IF (Uds_s.status = 1) THEN
	IF (Uds_s.status = 1 AND Uds_s.UdsTx.dataSize > 0) THEN
		IF (Uds_s.UdsTx.dataSize = Uds_s.UdsTx.data[1]) THEN (*send sf or ff*)
			IF (Uds_s.UdsTx.dataSize <= 7) THEN (*sf*)
				FOR y := 1 TO 8 DO
					tempCanSendBuff[y] := Uds_s.UdsTx.data[y];
				END_FOR
				IF (Uds_s.UdsTx.data[2] = 16#30) THEN
				can_sendDatabox(0, 42, Uds_s.UdsTx.dataSize, ADR(tempCanSendBuff) + 1);
				ELSE
				can_sendDatabox(0, 42, Uds_s.UdsTx.dataSize + 1, ADR(tempCanSendBuff));
				END_IF
				Uds_s.UdsTx.dataSize := 0;
				Uds_s.UdsTx.data[1] := 0;
			ELSE (*ff*)
				bytesTxFf[1] := 16#10;
				bytesTxFf[2] := Uds_s.UdsTx.data[1];
				FOR y := 3 TO 8 DO
					bytesTxFf[y] := Uds_s.UdsTx.data[y - 1];
				END_FOR
				Uds_s.UdsTx.data[1] := Uds_s.UdsTx.data[1] - 6;
				can_sendDatabox(0, 42, 8, ADR(bytesTxFf));
			END_IF
			Uds_s.status := 0;
		ELSIF (Uds_s.UdsTx.dataSize > Uds_s.UdsTx.data[1]) THEN (*cf*)
			startIndex := Uds_s.UdsTx.dataSize - Uds_s.UdsTx.data[1];
			bytesTxCf[1] := 16#20 + ((startIndex + 1) / 7) MOD 10;
			FOR txCfIdx := 2 TO 8 DO
				bytesTxCf[txCfIdx] := Uds_s.UdsTx.data[startIndex + txCfIdx];
				Uds_s.UdsTx.data[1] := Uds_s.UdsTx.data[1] - 1;
				IF (Uds_s.UdsTx.data[1] = 0) THEN
					EXIT;
				END_IF
			END_FOR
			IF (txCfIdx > 8) THEN
				txCfIdx := 8;
			END_IF
			can_sendDatabox(0, 42, txCfIdx, ADR(bytesTxCf));
			IF (Uds_s.UdsTx.data[1] = 0) THEN
				Uds_s.status := 0;
				Uds_s.UdsTx.dataSize := 0;
				Uds_s.UdsTx.data[1] := 0;
			END_IF
		END_IF
		Uds_s.tester := 0;
	END_IF
END_IF

IF (Uds_s.status = 0 AND Uds_s.UdsRx.data[1] = Uds_s.UdsRx.dataSize AND Uds_s.UdsRx.dataSize > 0) THEN
	Uds();
	Uds_s.UdsRx.dataSize := 0;
	Uds_s.UdsRx.data[1] := 0;
	Uds_s.status := 1;
END_IF
END_PROGRAM

(* POU Uds/Uds, ST *)
PROGRAM Uds
VAR
END_VAR
CASE Uds_s.UdsRx.data[2] OF
	16#10: UdsSrvDsc();
(*
	16#11: UdsSrvRst();*)
	16#14: UdsSrvClrDiagcInfo();

	16#19: UdsSrvReadDtcInfo();

	16#22: UdsSrvReadDataById();
(*
	16#23: UdsSrvReadMemByAddr();
	16#27: UdsSrvSecuAcs();*)
	16#2E: UdsSrvWriteDataById();
	(*16#31: UdsSrvRoutineCtrl();
	16#3D: UdsSrvWrMemByAddr();*)
	16#3E: UdsSrvTesterPresent();

ELSE
	UdsSrvNotSupported();
END_CASE;
END_PROGRAM

(* POU Uds/UdsSrvDsc, ST *)
PROGRAM UdsSrvDsc
VAR
END_VAR
IF (Uds_s.UdsRx.dataSize = 2 AND (Uds_s.UdsRx.data[3] = 16#01 OR Uds_s.UdsRx.data[3] = 16#03)) THEN
	Uds_s.sessionType := Uds_s.UdsRx.data[3];
	Uds_s.activeAccessLevel_u8 := LID_DevelopmentSession_DU8;(*LID_DefaultSession_DU8;*)
	Uds_s.UdsTx.dataSize := 6;
	Uds_s.UdsTx.data[1] := Uds_s.UdsTx.dataSize;
	Uds_s.UdsTx.data[2] := 16#50;
	Uds_s.UdsTx.data[3] := Uds_s.sessionType;
	Uds_s.UdsTx.data[4] := 16#00;
	Uds_s.UdsTx.data[5] := 16#96;
	Uds_s.UdsTx.data[6] := 16#01;
	Uds_s.UdsTx.data[7] := 16#F4;
ELSE
	UdsSrvNotSupported(); (*Temp solution, throw 7F error*)
END_IF
END_PROGRAM

(* POU Uds/UdsSrvNotSupported, ST *)
PROGRAM UdsSrvNotSupported
VAR
END_VAR
Uds_s.UdsTx.dataSize := 3;
Uds_s.UdsTx.data[1] := Uds_s.UdsTx.dataSize;
Uds_s.UdsTx.data[2] := 16#7F;
Uds_s.UdsTx.data[3] := Uds_s.UdsRx.data[3];
Uds_s.UdsTx.data[4] := 16#11;
END_PROGRAM

(* POU Uds/UdsSrvClrDiagcInfo, ST *)
PROGRAM UdsSrvClrDiagcInfo
VAR
	groupOfDtc : UDINT;
END_VAR
IF (Uds_s.UdsRx.dataSize = 4) THEN
	groupOfDtc := SHL(USINT_TO_UDINT(Uds_s.UdsRx.data[3]), 16);
	groupOfDtc := groupOfDtc + SHL(USINT_TO_UDINT(Uds_s.UdsRx.data[4]), 8);
	groupOfDtc := groupOfDtc + Uds_s.UdsRx.data[5];
	IF (groupOfDtc = 16#FFFFFF) THEN
		sys_enterCriticalSection();
		sys_delActiveErrors();
		sys_delSavedErrors();
		sys_leaveCriticalSection();
	END_IF
END_IF
END_PROGRAM

(* POU Uds/UdsSrvReadDtcInfo, ST *)
PROGRAM UdsSrvReadDtcInfo
VAR
	numSavedErr_u16        : UINT;
	numActvErr_u16         : UINT;
	numActvAndSavedErr_u16 : UINT;
	numErr_u16             : UINT;
	errData_s              : ErrorData_ts;
	idx_u16                : UINT;
	cntDtc_u16             : UINT;

	dtc_u32                : UDINT;
	dtcHB_u8               : USINT;
	dtcMB_u8               : USINT;
	dtcLB_u8               : USINT;

	buf_au8                : ARRAY[1..250] OF USINT; (*data without SID*)
	bufLength_u8           : USINT; (*actual data size*)
	i                      : USINT;
	idxErr_u8				  : USINT;
END_VAR
Uds_s.UdsTx.data[1] := 0;
IF (Uds_s.UdsRx.dataSize = 3) THEN
   IF (Uds_s.UdsRx.data[3] = 1) THEN
      sys_enterCriticalSection();
      IF (Uds_s.UdsRx.data[4] = 1) THEN
         numActvErr_u16 := sys_getNumActiveErrors();
      ELSIF (Uds_s.UdsRx.data[4] = 8) THEN
         numSavedErr_u16 := sys_getNumSavedErrors();
      END_IF
			IF (Uds_s.UdsRx.data[5] = 9) THEN
				WHILE(TRUE) DO
					numErr_u16 := sys_getSavedErrors( ADR(errData_s), idx_u16, 1);
				   IF numErr_u16 <> 1 THEN
					   EXIT;
				   END_IF

				   IF sys_testError(errData_s.Code_u16, errData_s.Param_u8) <> 0 THEN
					   numActvAndSavedErr_u16 := numActvAndSavedErr_u16 + 1;
				   END_IF
				   idx_u16 := idx_u16 + 1;
			   END_WHILE
			END_IF
		sys_leaveCriticalSection();
		IF ((numSavedErr_u16 + numActvErr_u16) >= numActvAndSavedErr_u16) THEN
			cntDtc_u16 := numSavedErr_u16 + numActvErr_u16 - numActvAndSavedErr_u16;
		ELSE
		   cntDtc_u16 := numSavedErr_u16 + numActvErr_u16;
	   END_IF

		Uds_s.UdsTx.data[1] := Uds_s.UdsTx.data[1] + 1;
		Uds_s.UdsTx.data[Uds_s.UdsTx.data[1] + 1 ] := Uds_s.UdsRx.data[2] + 16#40;
		Uds_s.UdsTx.data[1] := Uds_s.UdsTx.data[1] + 1;
		Uds_s.UdsTx.data[Uds_s.UdsTx.data[1] + 1 ] := Uds_s.UdsRx.data[3];
		Uds_s.UdsTx.data[1] := Uds_s.UdsTx.data[1] + 1;
		Uds_s.UdsTx.data[Uds_s.UdsTx.data[1] + 1 ] := Uds_s.UdsRx.data[4];
		Uds_s.UdsTx.data[1] := Uds_s.UdsTx.data[1] + 1;
		Uds_s.UdsTx.data[Uds_s.UdsTx.data[1] + 1 ] := Uds_s.UdsRx.data[5];
		Uds_s.UdsTx.data[1] := Uds_s.UdsTx.data[1] + 1;
		Uds_s.UdsTx.data[Uds_s.UdsTx.data[1] + 1 ] := UINT_TO_USINT(SHR(cntDtc_u16, 8));
		Uds_s.UdsTx.data[1] := Uds_s.UdsTx.data[1] + 1;
		Uds_s.UdsTx.data[Uds_s.UdsTx.data[1] + 1 ] := UINT_TO_USINT(cntDtc_u16);
	ELSIF (Uds_s.UdsRx.data[3] = 2) THEN
		sys_enterCriticalSection();
		IF (Uds_s.UdsRx.data[4] = 1) THEN (*read active errors codes*)
		Uds_s.UdsTx.data[1] := Uds_s.UdsTx.data[1] + 1;
		Uds_s.UdsTx.data[Uds_s.UdsTx.data[1] + 1 ] := Uds_s.UdsRx.data[2] + 16#40;
			WHILE(TRUE) DO
				numErr_u16 := sys_getActiveErrors( ADR(errData_s), idx_u16, 1);
				IF numErr_u16 <> 1 THEN
					EXIT;
				END_IF
				dtc_u32 := SHL(UINT_TO_UDINT(errData_s.Code_u16), 8) + errData_s.Param_u8;
				dtcHB_u8 := UDINT_TO_USINT(SHR(dtc_u32, 16));
				dtcMB_u8 := UDINT_TO_USINT(SHR(dtc_u32, 8));
				dtcLB_u8 := UDINT_TO_USINT(dtc_u32);
				(*FOR i:=0 TO cntDtc_u16 DO
				 ; (*check existing errors in buffer, 443 line in UdsReadDtcInfo.c*)
				END_FOR*)

				Uds_s.UdsTx.data[1] := Uds_s.UdsTx.data[1] + 1;
				Uds_s.UdsTx.data[Uds_s.UdsTx.data[1] + 1 ] := dtcHB_u8;
				Uds_s.UdsTx.data[1] := Uds_s.UdsTx.data[1] + 1;
				Uds_s.UdsTx.data[Uds_s.UdsTx.data[1] + 1 ] := dtcHB_u8; (*high byte*)
				Uds_s.UdsTx.data[1] := Uds_s.UdsTx.data[1] + 1;
				Uds_s.UdsTx.data[Uds_s.UdsTx.data[1] + 1 ] := dtcMB_u8; (*middle byte*)
				Uds_s.UdsTx.data[1] := Uds_s.UdsTx.data[1] + 1;
				Uds_s.UdsTx.data[Uds_s.UdsTx.data[1] + 1 ] := dtcLB_u8; (*low byte*)
				Uds_s.UdsTx.data[1] := Uds_s.UdsTx.data[1] + 1;
				Uds_s.UdsTx.data[Uds_s.UdsTx.data[1] + 1 ] := Uds_s.UdsRx.data[4];
				idx_u16 := idx_u16 + 1;
			END_WHILE
		ELSIF (Uds_s.UdsRx.data[4] = 8) THEN (*read saved errors codes*)
			;
      END_IF
		sys_leaveCriticalSection();
	END_IF


(*ELSE
   UdsSrvNotSupported();*)
END_IF
END_PROGRAM

(* POU Uds/UdsSrvReadDataById, ST *)
PROGRAM UdsSrvReadDataById
VAR
	didus : UINT;
END_VAR
IF (Uds_s.UdsRx.dataSize > 0 AND Uds_s.UdsRx.data[1] > 0) THEN
	didus := Uds_s.UdsRx.data[3];
	didus := SHL(didus, 8);
	didus := didus + Uds_s.UdsRx.data[4];

	CASE didus OF
		16#0000..16#1FFF:
			UdsGetParameters(did := didus);
		16#2000..16#21FF:
			UdsGetProcessData(did := didus);
		16#2200:
			UdsGetParameterMenuNames();
		16#2201..16#2400:
			UdsGetParameterSubMenuNames(did := didus);
		16#2401:
			UdsGetProcessGroupNames();
		16#2402:
			UdsGetUnitCodes();
		16#2403:
			UdsGetListDescriptions() ;
		16#2404:
			UdsGetErrors(errorType := 0);(*saved errors*)
		16#2405:
			UdsGetErrors(errorType := 1);(*active errors*)
		16#277F..16#4068:(*default uds DIDs for writing value/reading parameter value*)
			UdsDidAcsPrm(did := didus, flgWrDid := 0);
		16#4E2B..16#4F68:(*default uds DIDs for reading proccess value*)
			UdsDidAcsProcVal();
	ELSE
		UdsSrvNotSupported(); (*Temp solution, throw 7F error*)
	END_CASE;
END_IF
END_PROGRAM

(* POU Uds/UdsSrvReadDataByIdServices/UdsGetParameters, ST *)
PROGRAM UdsGetParameters

VAR_INPUT
    did: UINT;
END_VAR

VAR
	startIndex: USINT := 1;

	menuNumber: USINT;
	subMenuNumber: USINT;
	parameterNumber: USINT;
	nonEmptyParametersCount: USINT;

	parameterCounter: USINT;
	numberOfParameters: USINT;
	parameterNameLength : USINT;

	tempCounter: USINT;
	currentValue: UINT;
END_VAR
menuNumber := UINT_TO_BYTE(SHR(did, 7)) AND 16#3F;
menuNumber := menuNumber + 1;
subMenuNumber := UINT_TO_BYTE(SHR(did, 4)) AND 16#07;
subMenuNumber := subMenuNumber + 1;
parameterNumber := UINT_TO_BYTE(did) AND 16#0F;
parameterNumber :=parameterNumber + 1;
Uds_s.UdsTx.data[1] := 0;

Uds_s.UdsTx.data[1] := Uds_s.UdsTx.data[1] + 1;
Uds_s.UdsTx.data[Uds_s.UdsTx.data[1] + 1 ] := Uds_s.UdsRx.data[2] + 16#40;

IF (LEN(PrmData.ParameterMenus_as[menuNumber].MenuName_as8) > 0 AND LEN(PrmData.ParameterMenus_as[menuNumber].ParameterGroup_as[subMenuNumber].GroupName_as8) > 0) THEN
	 numberOfParameters := 8;
	IF(parameterNumber < 16#08) THEN
		startIndex := parameterNumber;
		numberOfParameters := parameterNumber;
	END_IF

	FOR parameterCounter := startIndex TO numberOfParameters DO
		parameterNameLength := INT_TO_USINT(LEN(PrmData.ParameterMenus_as[menuNumber].ParameterGroup_as[subMenuNumber].Param_as[parameterCounter].ParameterName_as8));
		IF (parameterNameLength > 0) THEN
			nonEmptyParametersCount := nonEmptyParametersCount + 1;
		END_IF
	END_FOR

	Uds_s.UdsTx.data[1] := Uds_s.UdsTx.data[1] + 1;
	Uds_s.UdsTx.data[Uds_s.UdsTx.data[1] + 1] := nonEmptyParametersCount;

	FOR parameterCounter := startIndex TO numberOfParameters DO
		parameterNameLength := INT_TO_USINT(LEN(PrmData.ParameterMenus_as[menuNumber].ParameterGroup_as[subMenuNumber].Param_as[parameterCounter].ParameterName_as8));
		IF (parameternameLength > 0) THEN
			Uds_s.UdsTx.data[1] := Uds_s.UdsTx.data[1] + 1;
			Uds_s.UdsTx.data[Uds_s.UdsTx.data[1] + 1] := parameterCounter - 1;

			IF (PrmData.ParameterMenus_as[menuNumber].ParameterGroup_as[subMenuNumber].Param_as[parameterCounter].AccesslevelCode_u8 <= Uds_s.activeAccessLevel_u8) THEN
				FOR tempCounter := 1 TO parameterNameLength DO
					Uds_s.UdsTx.data[1] := Uds_s.UdsTx.data[1] + 1;
					Uds_s.UdsTx.data[Uds_s.UdsTx.data[1] + 1] := BYTE_TO_USINT(CHARCODE(MID(PrmData.ParameterMenus_as[menuNumber].ParameterGroup_as[subMenuNumber].Param_as[parameterCounter].ParameterName_as8, 1, tempCounter)));
				END_FOR

				Uds_s.UdsTx.data[1] := Uds_s.UdsTx.data[1] + 1;
				Uds_s.UdsTx.data[Uds_s.UdsTx.data[1] + 1] := 0;

				currentValue := ree_getValue(PrmData.ParameterMenus_as[menuNumber].ParameterGroup_as[subMenuNumber].Param_as[parameterCounter].EEPROMAddress_s.Page_u8, PrmData.ParameterMenus_as[menuNumber].ParameterGroup_as[subMenuNumber].Param_as[parameterCounter].EEPROMAddress_s.IntIndex_u8);

				Uds_s.UdsTx.data[1] := Uds_s.UdsTx.data[1] + 1;
				Uds_s.UdsTx.data[Uds_s.UdsTx.data[1] + 1] := UINT_TO_USINT(SHR(currentValue, 8));
				Uds_s.UdsTx.data[1] := Uds_s.UdsTx.data[1] + 1;
				Uds_s.UdsTx.data[Uds_s.UdsTx.data[1] + 1] := UINT_TO_USINT(currentValue);

				Uds_s.UdsTx.data[1] := Uds_s.UdsTx.data[1] + 1;
				Uds_s.UdsTx.data[Uds_s.UdsTx.data[1] + 1] := INT_TO_USINT(SHR(PrmData.ParameterMenus_as[menuNumber].ParameterGroup_as[subMenuNumber].Param_as[parameterCounter].Multiplier_s16, 8));
				Uds_s.UdsTx.data[1] := Uds_s.UdsTx.data[1] + 1;
				Uds_s.UdsTx.data[Uds_s.UdsTx.data[1] + 1] := INT_TO_USINT(PrmData.ParameterMenus_as[menuNumber].ParameterGroup_as[subMenuNumber].Param_as[parameterCounter].Multiplier_s16);

				Uds_s.UdsTx.data[1] := Uds_s.UdsTx.data[1] + 1;
				Uds_s.UdsTx.data[Uds_s.UdsTx.data[1] + 1] := INT_TO_USINT(SHR(PrmData.ParameterMenus_as[menuNumber].ParameterGroup_as[subMenuNumber].Param_as[parameterCounter].Divisor_s16, 8));
				Uds_s.UdsTx.data[1] := Uds_s.UdsTx.data[1] + 1;
				Uds_s.UdsTx.data[Uds_s.UdsTx.data[1] + 1] := INT_TO_USINT(PrmData.ParameterMenus_as[menuNumber].ParameterGroup_as[subMenuNumber].Param_as[parameterCounter].Divisor_s16);

				Uds_s.UdsTx.data[1] := Uds_s.UdsTx.data[1] + 1;
				Uds_s.UdsTx.data[Uds_s.UdsTx.data[1] + 1] := UINT_TO_USINT(SHR(PrmData.ParameterMenus_as[menuNumber].ParameterGroup_as[subMenuNumber].Param_as[parameterCounter].NumberOfDigits_u16, 8));
				Uds_s.UdsTx.data[1] := Uds_s.UdsTx.data[1] + 1;
				Uds_s.UdsTx.data[Uds_s.UdsTx.data[1] + 1] := UINT_TO_USINT(PrmData.ParameterMenus_as[menuNumber].ParameterGroup_as[subMenuNumber].Param_as[parameterCounter].NumberOfDigits_u16);

				Uds_s.UdsTx.data[1] := Uds_s.UdsTx.data[1] + 1;
				Uds_s.UdsTx.data[Uds_s.UdsTx.data[1] + 1] := PrmData.ParameterMenus_as[menuNumber].ParameterGroup_as[subMenuNumber].Param_as[parameterCounter].ParameterType_u8;

				Uds_s.UdsTx.data[1] := Uds_s.UdsTx.data[1] + 1;
				Uds_s.UdsTx.data[Uds_s.UdsTx.data[1] + 1] := INT_TO_USINT(SHR(PrmData.ParameterMenus_as[menuNumber].ParameterGroup_as[subMenuNumber].Param_as[parameterCounter].attr1_u, 8));
				Uds_s.UdsTx.data[1] := Uds_s.UdsTx.data[1] + 1;
				Uds_s.UdsTx.data[Uds_s.UdsTx.data[1] + 1] := INT_TO_USINT(PrmData.ParameterMenus_as[menuNumber].ParameterGroup_as[subMenuNumber].Param_as[parameterCounter].attr1_u);

				Uds_s.UdsTx.data[1] := Uds_s.UdsTx.data[1] + 1;
				Uds_s.UdsTx.data[Uds_s.UdsTx.data[1] + 1] := INT_TO_USINT(SHR(PrmData.ParameterMenus_as[menuNumber].ParameterGroup_as[subMenuNumber].Param_as[parameterCounter].attr2_u, 8));
				Uds_s.UdsTx.data[1] := Uds_s.UdsTx.data[1] + 1;
				Uds_s.UdsTx.data[Uds_s.UdsTx.data[1] + 1] := INT_TO_USINT(PrmData.ParameterMenus_as[menuNumber].ParameterGroup_as[subMenuNumber].Param_as[parameterCounter].attr2_u);

				Uds_s.UdsTx.data[1] := Uds_s.UdsTx.data[1] + 1;
				Uds_s.UdsTx.data[Uds_s.UdsTx.data[1] + 1] := UINT_TO_USINT(SHR(PrmData.ParameterMenus_as[menuNumber].ParameterGroup_as[subMenuNumber].Param_as[parameterCounter].attr3_u, 8));
				Uds_s.UdsTx.data[1] := Uds_s.UdsTx.data[1] + 1;
				Uds_s.UdsTx.data[Uds_s.UdsTx.data[1] + 1] := UINT_TO_USINT(PrmData.ParameterMenus_as[menuNumber].ParameterGroup_as[subMenuNumber].Param_as[parameterCounter].attr3_u);

				Uds_s.UdsTx.data[1] := Uds_s.UdsTx.data[1] + 1;
				Uds_s.UdsTx.data[Uds_s.UdsTx.data[1] + 1] := INT_TO_USINT(SHR(PrmData.ParameterMenus_as[menuNumber].ParameterGroup_as[subMenuNumber].Param_as[parameterCounter].attr4_u, 8));
				Uds_s.UdsTx.data[1] := Uds_s.UdsTx.data[1] + 1;
				Uds_s.UdsTx.data[Uds_s.UdsTx.data[1] + 1] := INT_TO_USINT(PrmData.ParameterMenus_as[menuNumber].ParameterGroup_as[subMenuNumber].Param_as[parameterCounter].attr4_u);

				Uds_s.UdsTx.data[1] := Uds_s.UdsTx.data[1] + 1;
				Uds_s.UdsTx.data[Uds_s.UdsTx.data[1] + 1] := PrmData.ParameterMenus_as[menuNumber].ParameterGroup_as[subMenuNumber].Param_as[parameterCounter].UnitCode_au8;

				Uds_s.UdsTx.data[1] := Uds_s.UdsTx.data[1] + 1;
				Uds_s.UdsTx.data[Uds_s.UdsTx.data[1] + 1] := PrmData.ParameterMenus_as[menuNumber].ParameterGroup_as[subMenuNumber].Param_as[parameterCounter].EEPROMAddress_s.IntIndex_u8;

				Uds_s.UdsTx.data[1] := Uds_s.UdsTx.data[1] + 1;
				Uds_s.UdsTx.data[Uds_s.UdsTx.data[1] + 1] := PrmData.ParameterMenus_as[menuNumber].ParameterGroup_as[subMenuNumber].Param_as[parameterCounter].EEPROMAddress_s.Page_u8;

				Uds_s.UdsTx.data[1] := Uds_s.UdsTx.data[1] + 1;
				Uds_s.UdsTx.data[Uds_s.UdsTx.data[1] + 1] := PrmData.ParameterMenus_as[menuNumber].ParameterGroup_as[subMenuNumber].Param_as[parameterCounter].AccesslevelCode_u8;

				IF (parameterCounter < 8 AND LEN(PrmData.ParameterMenus_as[menuNumber].ParameterGroup_as[subMenuNumber].Param_as[parameterCounter + 1].ParameterName_as8) + 24 > (255 - Uds_s.UdsTx.data[1])) THEN
					EXIT;
				END_IF

			ELSE
				Uds_s.UdsTx.data[1] := Uds_s.UdsTx.data[1] + 1;
				Uds_s.UdsTx.data[Uds_s.UdsTx.data[1] + 1] := 0;
			END_IF
		END_IF
	END_FOR

	IF (parameterCounter = numberOfParameters + 1) THEN
		startIndex := 1;
	ELSE
		startIndex := parameterCounter + 1;
	END_IF
END_IF
Uds_s.UdsTx.dataSize := Uds_s.UdsTx.data[1];
END_PROGRAM

(* POU Autocode/PrmData, ST *)
PROGRAM PrmData
(*********************************************)
(*  DON'T MAKE ANY CHANGES TO THIS PROGRAM!! *)
(*     FILE WAS AUTOMATICALLY GENERATED!!    *)
(*********************************************)

VAR
END_VAR
VAR CONSTANT

(**)
(*********************************************)
nrPrmMenus_u8          : USINT := 5;

(*********************************************)
(* Parameters Tree *)
(*********************************************)

ParameterMenus_as      : ARRAY [1..5] OF ParameterMenu_ts := 

   (*********************************************)
   (* parameter menu 1 - up to 8 groups can be defined here *)
   (*********************************************)
   (
      MenuName_as8        := 'Menu 1',

      ParameterGroup_as   := 

      (*********************************************)
      (* parameter group 1.1 - up to 8 parameters can be defined here *)
      (*********************************************)
      (
         GroupName_as8   := 'Basic',

         Param_as        := 

         (*********************************************)
         (* parameter 1.1.1 *)
         (*********************************************)
         (
            ParameterName_as8    := 'List test 1',
            ParameterType_u8     := 0,
            attr1_u              := 0,
            attr2_u              := 2,
            UnitCode_au8         := 0,
            AccesslevelCode_u8   := 129,
            attr4_u              := 0,
            EEPROMAddress_s      := (Page_u8 := 3, IntIndex_u8 := 22)
         ),

         (*********************************************)
         (* parameter 1.1.2 *)
         (*********************************************)
         (
            ParameterName_as8    := 'Input_to_Output_Mode',
            ParameterType_u8     := 7,
            attr1_u              := 0,
            attr2_u              := 2,
            UnitCode_au8         := 0,
            AccesslevelCode_u8   := 129,
            attr4_u              := 0,
            EEPROMAddress_s      := (Page_u8 := 3, IntIndex_u8 := 2)
         ),

         (*********************************************)
         (* parameter 1.1.3 *)
         (*********************************************)
         (
         ),

         (*********************************************)
         (* parameter 1.1.4 *)
         (*********************************************)
         (
            ParameterName_as8    := 'Test parameter new',
            ParameterType_u8     := 7,
            attr1_u              := 0,
            attr2_u              := 2,
            UnitCode_au8         := 0,
            AccesslevelCode_u8   := 129,
            attr4_u              := 0,
            EEPROMAddress_s      := (Page_u8 := 3, IntIndex_u8 := 5)
         ),

         (*********************************************)
         (* parameter 1.1.5 *)
         (*********************************************)
         (
         ),

         (*********************************************)
         (* parameter 1.1.6 *)
         (*********************************************)
         (
            ParameterName_as8    := 'Test_parameter',
            ParameterType_u8     := 7,
            attr1_u              := 0,
            attr2_u              := 2,
            UnitCode_au8         := 0,
            AccesslevelCode_u8   := 129,
            attr4_u              := 0,
            EEPROMAddress_s      := (Page_u8 := 3, IntIndex_u8 := 3)
         ),

         (*********************************************)
         (* parameter 1.1.7 *)
         (*********************************************)
         (
         ),

         (*********************************************)
         (* parameter 1.1.8 *)
         (*********************************************)
         (
            ParameterName_as8    := 'Test_params',
            ParameterType_u8     := 7,
            attr1_u              := 0,
            attr2_u              := 2,
            UnitCode_au8         := 0,
            AccesslevelCode_u8   := 129,
            attr4_u              := 0,
            EEPROMAddress_s      := (Page_u8 := 3, IntIndex_u8 := 4)
         )

      ),

      (*********************************************)
      (* parameter group 1.2 - up to 8 parameters can be defined here *)
      (*********************************************)
      (
         GroupName_as8   := 'Test Type',

         Param_as        := 

         (*********************************************)
         (* parameter 1.2.1 *)
         (*********************************************)
         (
            ParameterName_as8    := 'Trimming type',
            ParameterType_u8     := 5,
            attr1_u              := 0,
            attr2_u              := 511,
            UnitCode_au8         := 0,
            AccesslevelCode_u8   := 129,
            attr4_u              := 0,
            EEPROMAddress_s      := (Page_u8 := 3, IntIndex_u8 := 50)
         ),

         (*********************************************)
         (* parameter 1.2.2 *)
         (*********************************************)
         (
            ParameterName_as8    := 'Analog type',
            ParameterType_u8     := 8,
            attr1_u              := 53,
            UnitCode_au8         := 0,
            AccesslevelCode_u8   := 129,
            attr4_u              := 249,
            EEPROMAddress_s      := (Page_u8 := 3, IntIndex_u8 := 51)
         ),

         (*********************************************)
         (* parameter 1.2.3 *)
         (*********************************************)
         (
            ParameterName_as8    := 'Curve Type',
            ParameterType_u8     := 6,
            attr1_u              := 66,
            attr2_u              := 67,
            attr3_u              := 3000,
            UnitCode_au8         := 0,
            AccesslevelCode_u8   := 129,
            attr4_u              := 245,
            EEPROMAddress_s      := (Page_u8 := 3, IntIndex_u8 := 52)
         ),

         (*********************************************)
         (* parameter 1.2.4 *)
         (*********************************************)
         (
            ParameterName_as8    := 'Function Type',
            ParameterType_u8     := 9,
            attr1_u              := 248,
            attr2_u              := 254,
            attr3_u              := 248,
            UnitCode_au8         := 0,
            AccesslevelCode_u8   := 129,
            attr4_u              := 248,
            EEPROMAddress_s      := (Page_u8 := 3, IntIndex_u8 := 53)
         ),

         (*********************************************)
         (* parameter 1.2.5 *)
         (*********************************************)
         (
            ParameterName_as8    := 'Percent Type',
            ParameterType_u8     := 0,
            attr1_u              := 0,
            attr2_u              := 1000,
            attr3_u              := 10,
            UnitCode_au8         := 1,
            Multiplier_s16       := 1,
            Divisor_s16          := 1,
            NumberOfDigits_u16   := 0,
            AccesslevelCode_u8   := 129,
            attr4_u              := 0,
            EEPROMAddress_s      := (Page_u8 := 3, IntIndex_u8 := 54)
         ),

         (*********************************************)
         (* parameter 1.2.6 *)
         (*********************************************)
         (
            ParameterName_as8    := 'Ramp Type',
            ParameterType_u8     := 0,
            attr1_u              := 0,
            attr2_u              := 100,
            attr3_u              := 10,
            UnitCode_au8         := 1,
            Multiplier_s16       := 1,
            Divisor_s16          := 1,
            NumberOfDigits_u16   := 0,
            AccesslevelCode_u8   := 129,
            attr4_u              := 0,
            EEPROMAddress_s      := (Page_u8 := 3, IntIndex_u8 := 55)
         ),

         (*********************************************)
         (* parameter 1.2.7 *)
         (*********************************************)
         (
            ParameterName_as8    := 'Switch Type',
            ParameterType_u8     := 4,
            UnitCode_au8         := 0,
            AccesslevelCode_u8   := 129,
            attr4_u              := 1,
            EEPROMAddress_s      := (Page_u8 := 3, IntIndex_u8 := 56)
         ),

         (*********************************************)
         (* parameter 1.2.8 *)
         (*********************************************)
         (
            ParameterName_as8    := 'List Type',
            ParameterType_u8     := 7,
            attr1_u              := 3,
            attr2_u              := 2,
            UnitCode_au8         := 0,
            AccesslevelCode_u8   := 129,
            attr4_u              := 0,
            EEPROMAddress_s      := (Page_u8 := 3, IntIndex_u8 := 57)
         )

      ),

      (*********************************************)
      (* parameter group 1.3 - up to 8 parameters can be defined here *)
      (*********************************************)
      (
         GroupName_as8   := 'Test Number',

         Param_as        := 

         (*********************************************)
         (* parameter 1.3.1 *)
         (*********************************************)
         (
            ParameterName_as8    := 'Number test 1',
            ParameterType_u8     := 0,
            attr1_u              := 0,
            attr2_u              := 30000,
            attr3_u              := 1,
            UnitCode_au8         := 4,
            Multiplier_s16       := 1,
            Divisor_s16          := 1,
            NumberOfDigits_u16   := 0,
            AccesslevelCode_u8   := 129,
            attr4_u              := 0,
            EEPROMAddress_s      := (Page_u8 := 3, IntIndex_u8 := 14)
         ),

         (*********************************************)
         (* parameter 1.3.2 *)
         (*********************************************)
         (
            ParameterName_as8    := 'Number test 2',
            ParameterType_u8     := 0,
            attr1_u              := 0,
            attr2_u              := 30000,
            attr3_u              := 1,
            UnitCode_au8         := 4,
            Multiplier_s16       := 1,
            Divisor_s16          := 1,
            NumberOfDigits_u16   := 0,
            AccesslevelCode_u8   := 129,
            attr4_u              := 0,
            EEPROMAddress_s      := (Page_u8 := 3, IntIndex_u8 := 15)
         ),

         (*********************************************)
         (* parameter 1.3.3 *)
         (*********************************************)
         (
            ParameterName_as8    := 'Number test 3',
            ParameterType_u8     := 0,
            attr1_u              := 0,
            attr2_u              := 30000,
            attr3_u              := 1,
            UnitCode_au8         := 4,
            Multiplier_s16       := 1,
            Divisor_s16          := 1,
            NumberOfDigits_u16   := 0,
            AccesslevelCode_u8   := 129,
            attr4_u              := 0,
            EEPROMAddress_s      := (Page_u8 := 3, IntIndex_u8 := 16)
         ),

         (*********************************************)
         (* parameter 1.3.4 *)
         (*********************************************)
         (
            ParameterName_as8    := 'Number test 4',
            ParameterType_u8     := 0,
            attr1_u              := 0,
            attr2_u              := 30000,
            attr3_u              := 1,
            UnitCode_au8         := 4,
            Multiplier_s16       := 1,
            Divisor_s16          := 1,
            NumberOfDigits_u16   := 0,
            AccesslevelCode_u8   := 129,
            attr4_u              := 0,
            EEPROMAddress_s      := (Page_u8 := 3, IntIndex_u8 := 17)
         ),

         (*********************************************)
         (* parameter 1.3.5 *)
         (*********************************************)
         (
            ParameterName_as8    := 'Number test 5',
            ParameterType_u8     := 0,
            attr1_u              := 0,
            attr2_u              := 30000,
            attr3_u              := 1,
            UnitCode_au8         := 4,
            Multiplier_s16       := 1,
            Divisor_s16          := 1,
            NumberOfDigits_u16   := 0,
            AccesslevelCode_u8   := 129,
            attr4_u              := 0,
            EEPROMAddress_s      := (Page_u8 := 3, IntIndex_u8 := 18)
         ),

         (*********************************************)
         (* parameter 1.3.6 *)
         (*********************************************)
         (
            ParameterName_as8    := 'Number test 6',
            ParameterType_u8     := 0,
            attr1_u              := 0,
            attr2_u              := 30000,
            attr3_u              := 1,
            UnitCode_au8         := 4,
            Multiplier_s16       := 1,
            Divisor_s16          := 1,
            NumberOfDigits_u16   := 0,
            AccesslevelCode_u8   := 129,
            attr4_u              := 0,
            EEPROMAddress_s      := (Page_u8 := 3, IntIndex_u8 := 19)
         ),

         (*********************************************)
         (* parameter 1.3.7 *)
         (*********************************************)
         (
            ParameterName_as8    := 'Number test 7',
            ParameterType_u8     := 0,
            attr1_u              := 0,
            attr2_u              := 30000,
            attr3_u              := 1,
            UnitCode_au8         := 4,
            Multiplier_s16       := 1,
            Divisor_s16          := 1,
            NumberOfDigits_u16   := 0,
            AccesslevelCode_u8   := 129,
            attr4_u              := 0,
            EEPROMAddress_s      := (Page_u8 := 3, IntIndex_u8 := 20)
         ),

         (*********************************************)
         (* parameter 1.3.8 *)
         (*********************************************)
         (
            ParameterName_as8    := 'Number test 8',
            ParameterType_u8     := 0,
            attr1_u              := 0,
            attr2_u              := 30000,
            attr3_u              := 1,
            UnitCode_au8         := 4,
            Multiplier_s16       := 1,
            Divisor_s16          := 1,
            NumberOfDigits_u16   := 0,
            AccesslevelCode_u8   := 129,
            attr4_u              := 0,
            EEPROMAddress_s      := (Page_u8 := 3, IntIndex_u8 := 21)
         )

      ),

      (*********************************************)
      (* parameter group 1.4 - up to 8 parameters can be defined here *)
      (*********************************************)
      (








      ),

      (*********************************************)
      (* parameter group 1.5 - up to 8 parameters can be defined here *)
      (*********************************************)
      (








      ),

      (*********************************************)
      (* parameter group 1.6 - up to 8 parameters can be defined here *)
      (*********************************************)
      (








      ),

      (*********************************************)
      (* parameter group 1.7 - up to 8 parameters can be defined here *)
      (*********************************************)
      (








      ),

      (*********************************************)
      (* parameter group 1.8 - up to 8 parameters can be defined here *)
      (*********************************************)
      (








      )

   ),

   (*********************************************)
   (* parameter menu 2 - up to 8 groups can be defined here *)
   (*********************************************)
   (
      MenuName_as8        := 'Menu 2',

      ParameterGroup_as   := 

      (*********************************************)
      (* parameter group 2.1 - up to 8 parameters can be defined here *)
      (*********************************************)
      (
         GroupName_as8   := 'Output Cfg 1-8',

         Param_as        := 

         (*********************************************)
         (* parameter 2.1.1 *)
         (*********************************************)
         (
            ParameterName_as8    := 'Output Cfg 1',
            ParameterType_u8     := 7,
            attr1_u              := 1,
            attr2_u              := 2,
            UnitCode_au8         := 0,
            AccesslevelCode_u8   := 129,
            attr4_u              := 0,
            EEPROMAddress_s      := (Page_u8 := 3, IntIndex_u8 := 64)
         ),

         (*********************************************)
         (* parameter 2.1.2 *)
         (*********************************************)
         (
            ParameterName_as8    := 'Output Cfg 2',
            ParameterType_u8     := 7,
            attr1_u              := 1,
            attr2_u              := 2,
            UnitCode_au8         := 0,
            AccesslevelCode_u8   := 129,
            attr4_u              := 0,
            EEPROMAddress_s      := (Page_u8 := 3, IntIndex_u8 := 65)
         ),

         (*********************************************)
         (* parameter 2.1.3 *)
         (*********************************************)
         (
            ParameterName_as8    := 'Output Cfg 3',
            ParameterType_u8     := 7,
            attr1_u              := 1,
            attr2_u              := 2,
            UnitCode_au8         := 0,
            AccesslevelCode_u8   := 129,
            attr4_u              := 0,
            EEPROMAddress_s      := (Page_u8 := 3, IntIndex_u8 := 66)
         ),

         (*********************************************)
         (* parameter 2.1.4 *)
         (*********************************************)
         (
            ParameterName_as8    := 'Output Cfg 4',
            ParameterType_u8     := 7,
            attr1_u              := 1,
            attr2_u              := 2,
            UnitCode_au8         := 0,
            AccesslevelCode_u8   := 129,
            attr4_u              := 0,
            EEPROMAddress_s      := (Page_u8 := 3, IntIndex_u8 := 67)
         ),

         (*********************************************)
         (* parameter 2.1.5 *)
         (*********************************************)
         (
            ParameterName_as8    := 'Output Cfg 5',
            ParameterType_u8     := 7,
            attr1_u              := 1,
            attr2_u              := 2,
            UnitCode_au8         := 0,
            AccesslevelCode_u8   := 129,
            attr4_u              := 0,
            EEPROMAddress_s      := (Page_u8 := 3, IntIndex_u8 := 68)
         ),

         (*********************************************)
         (* parameter 2.1.6 *)
         (*********************************************)
         (
            ParameterName_as8    := 'Output Cfg 6',
            ParameterType_u8     := 7,
            attr1_u              := 1,
            attr2_u              := 2,
            UnitCode_au8         := 0,
            AccesslevelCode_u8   := 129,
            attr4_u              := 0,
            EEPROMAddress_s      := (Page_u8 := 3, IntIndex_u8 := 69)
         ),

         (*********************************************)
         (* parameter 2.1.7 *)
         (*********************************************)
         (
            ParameterName_as8    := 'Output Cfg 7',
            ParameterType_u8     := 7,
            attr1_u              := 1,
            attr2_u              := 2,
            UnitCode_au8         := 0,
            AccesslevelCode_u8   := 129,
            attr4_u              := 0,
            EEPROMAddress_s      := (Page_u8 := 3, IntIndex_u8 := 70)
         ),

         (*********************************************)
         (* parameter 2.1.8 *)
         (*********************************************)
         (
            ParameterName_as8    := 'Output Cfg 8',
            ParameterType_u8     := 7,
            attr1_u              := 1,
            attr2_u              := 2,
            UnitCode_au8         := 0,
            AccesslevelCode_u8   := 129,
            attr4_u              := 0,
            EEPROMAddress_s      := (Page_u8 := 3, IntIndex_u8 := 71)
         )

      ),

      (*********************************************)
      (* parameter group 2.2 - up to 8 parameters can be defined here *)
      (*********************************************)
      (
         GroupName_as8   := 'Output Cfg 9-16',

         Param_as        := 

         (*********************************************)
         (* parameter 2.2.1 *)
         (*********************************************)
         (
            ParameterName_as8    := 'Output Cfg 9',
            ParameterType_u8     := 7,
            attr1_u              := 1,
            attr2_u              := 2,
            UnitCode_au8         := 0,
            AccesslevelCode_u8   := 129,
            attr4_u              := 0,
            EEPROMAddress_s      := (Page_u8 := 3, IntIndex_u8 := 72)
         ),

         (*********************************************)
         (* parameter 2.2.2 *)
         (*********************************************)
         (
            ParameterName_as8    := 'Output Cfg 10',
            ParameterType_u8     := 7,
            attr1_u              := 1,
            attr2_u              := 2,
            UnitCode_au8         := 0,
            AccesslevelCode_u8   := 129,
            attr4_u              := 0,
            EEPROMAddress_s      := (Page_u8 := 3, IntIndex_u8 := 73)
         ),

         (*********************************************)
         (* parameter 2.2.3 *)
         (*********************************************)
         (
            ParameterName_as8    := 'Output Cfg 11',
            ParameterType_u8     := 7,
            attr1_u              := 1,
            attr2_u              := 2,
            UnitCode_au8         := 0,
            AccesslevelCode_u8   := 129,
            attr4_u              := 0,
            EEPROMAddress_s      := (Page_u8 := 3, IntIndex_u8 := 74)
         ),

         (*********************************************)
         (* parameter 2.2.4 *)
         (*********************************************)
         (
            ParameterName_as8    := 'Output Cfg 12',
            ParameterType_u8     := 7,
            attr1_u              := 1,
            attr2_u              := 2,
            UnitCode_au8         := 0,
            AccesslevelCode_u8   := 129,
            attr4_u              := 0,
            EEPROMAddress_s      := (Page_u8 := 3, IntIndex_u8 := 75)
         ),

         (*********************************************)
         (* parameter 2.2.5 *)
         (*********************************************)
         (
            ParameterName_as8    := 'Output Cfg 13',
            ParameterType_u8     := 7,
            attr1_u              := 1,
            attr2_u              := 2,
            UnitCode_au8         := 0,
            AccesslevelCode_u8   := 129,
            attr4_u              := 0,
            EEPROMAddress_s      := (Page_u8 := 3, IntIndex_u8 := 76)
         ),

         (*********************************************)
         (* parameter 2.2.6 *)
         (*********************************************)
         (
            ParameterName_as8    := 'Output Cfg 14',
            ParameterType_u8     := 7,
            attr1_u              := 1,
            attr2_u              := 2,
            UnitCode_au8         := 0,
            AccesslevelCode_u8   := 129,
            attr4_u              := 0,
            EEPROMAddress_s      := (Page_u8 := 3, IntIndex_u8 := 77)
         ),

         (*********************************************)
         (* parameter 2.2.7 *)
         (*********************************************)
         (
            ParameterName_as8    := 'Output Cfg 15',
            ParameterType_u8     := 7,
            attr1_u              := 1,
            attr2_u              := 2,
            UnitCode_au8         := 0,
            AccesslevelCode_u8   := 129,
            attr4_u              := 0,
            EEPROMAddress_s      := (Page_u8 := 3, IntIndex_u8 := 78)
         ),

         (*********************************************)
         (* parameter 2.2.8 *)
         (*********************************************)
         (
            ParameterName_as8    := 'Output Cfg 16',
            ParameterType_u8     := 7,
            attr1_u              := 1,
            attr2_u              := 2,
            UnitCode_au8         := 0,
            AccesslevelCode_u8   := 129,
            attr4_u              := 0,
            EEPROMAddress_s      := (Page_u8 := 3, IntIndex_u8 := 79)
         )

      ),

      (*********************************************)
      (* parameter group 2.3 - up to 8 parameters can be defined here *)
      (*********************************************)
      (
         GroupName_as8   := 'Output Cfg 17-24',

         Param_as        := 

         (*********************************************)
         (* parameter 2.3.1 *)
         (*********************************************)
         (
            ParameterName_as8    := 'Output Cfg 17',
            ParameterType_u8     := 7,
            attr1_u              := 1,
            attr2_u              := 2,
            UnitCode_au8         := 0,
            AccesslevelCode_u8   := 129,
            attr4_u              := 0,
            EEPROMAddress_s      := (Page_u8 := 3, IntIndex_u8 := 80)
         ),

         (*********************************************)
         (* parameter 2.3.2 *)
         (*********************************************)
         (
            ParameterName_as8    := 'Output Cfg 18',
            ParameterType_u8     := 7,
            attr1_u              := 1,
            attr2_u              := 2,
            UnitCode_au8         := 0,
            AccesslevelCode_u8   := 129,
            attr4_u              := 0,
            EEPROMAddress_s      := (Page_u8 := 3, IntIndex_u8 := 81)
         ),

         (*********************************************)
         (* parameter 2.3.3 *)
         (*********************************************)
         (
            ParameterName_as8    := 'Output Cfg 19',
            ParameterType_u8     := 7,
            attr1_u              := 0,
            attr2_u              := 2,
            UnitCode_au8         := 0,
            AccesslevelCode_u8   := 129,
            attr4_u              := 0,
            EEPROMAddress_s      := (Page_u8 := 3, IntIndex_u8 := 82)
         ),

         (*********************************************)
         (* parameter 2.3.4 *)
         (*********************************************)
         (
            ParameterName_as8    := 'Output Cfg 20',
            ParameterType_u8     := 7,
            attr1_u              := 0,
            attr2_u              := 2,
            UnitCode_au8         := 0,
            AccesslevelCode_u8   := 129,
            attr4_u              := 0,
            EEPROMAddress_s      := (Page_u8 := 3, IntIndex_u8 := 83)
         ),

         (*********************************************)
         (* parameter 2.3.5 *)
         (*********************************************)
         (
            ParameterName_as8    := 'Output Cfg 21',
            ParameterType_u8     := 7,
            attr1_u              := 0,
            attr2_u              := 2,
            UnitCode_au8         := 0,
            AccesslevelCode_u8   := 129,
            attr4_u              := 0,
            EEPROMAddress_s      := (Page_u8 := 3, IntIndex_u8 := 84)
         ),

         (*********************************************)
         (* parameter 2.3.6 *)
         (*********************************************)
         (
            ParameterName_as8    := 'Output Cfg 22',
            ParameterType_u8     := 7,
            attr1_u              := 0,
            attr2_u              := 2,
            UnitCode_au8         := 0,
            AccesslevelCode_u8   := 129,
            attr4_u              := 0,
            EEPROMAddress_s      := (Page_u8 := 3, IntIndex_u8 := 85)
         ),

         (*********************************************)
         (* parameter 2.3.7 *)
         (*********************************************)
         (
            ParameterName_as8    := 'Output Cfg 23',
            ParameterType_u8     := 7,
            attr1_u              := 0,
            attr2_u              := 2,
            UnitCode_au8         := 0,
            AccesslevelCode_u8   := 129,
            attr4_u              := 0,
            EEPROMAddress_s      := (Page_u8 := 3, IntIndex_u8 := 86)
         ),

         (*********************************************)
         (* parameter 2.3.8 *)
         (*********************************************)
         (
            ParameterName_as8    := 'Output Cfg 24',
            ParameterType_u8     := 7,
            attr1_u              := 0,
            attr2_u              := 2,
            UnitCode_au8         := 0,
            AccesslevelCode_u8   := 129,
            attr4_u              := 0,
            EEPROMAddress_s      := (Page_u8 := 3, IntIndex_u8 := 87)
         )

      ),

      (*********************************************)
      (* parameter group 2.4 - up to 8 parameters can be defined here *)
      (*********************************************)
      (
         GroupName_as8   := 'Output Cfg 25-32',

         Param_as        := 

         (*********************************************)
         (* parameter 2.4.1 *)
         (*********************************************)
         (
            ParameterName_as8    := 'Output Cfg 25',
            ParameterType_u8     := 7,
            attr1_u              := 0,
            attr2_u              := 2,
            UnitCode_au8         := 0,
            AccesslevelCode_u8   := 129,
            attr4_u              := 0,
            EEPROMAddress_s      := (Page_u8 := 3, IntIndex_u8 := 88)
         ),

         (*********************************************)
         (* parameter 2.4.2 *)
         (*********************************************)
         (
            ParameterName_as8    := 'Output Cfg 26',
            ParameterType_u8     := 7,
            attr1_u              := 0,
            attr2_u              := 2,
            UnitCode_au8         := 0,
            AccesslevelCode_u8   := 129,
            attr4_u              := 0,
            EEPROMAddress_s      := (Page_u8 := 3, IntIndex_u8 := 89)
         ),

         (*********************************************)
         (* parameter 2.4.3 *)
         (*********************************************)
         (
            ParameterName_as8    := 'Output Cfg 27',
            ParameterType_u8     := 7,
            attr1_u              := 0,
            attr2_u              := 2,
            UnitCode_au8         := 0,
            AccesslevelCode_u8   := 129,
            attr4_u              := 0,
            EEPROMAddress_s      := (Page_u8 := 3, IntIndex_u8 := 90)
         ),

         (*********************************************)
         (* parameter 2.4.4 *)
         (*********************************************)
         (
            ParameterName_as8    := 'Output Cfg 28',
            ParameterType_u8     := 7,
            attr1_u              := 0,
            attr2_u              := 2,
            UnitCode_au8         := 0,
            AccesslevelCode_u8   := 129,
            attr4_u              := 0,
            EEPROMAddress_s      := (Page_u8 := 3, IntIndex_u8 := 91)
         ),

         (*********************************************)
         (* parameter 2.4.5 *)
         (*********************************************)
         (
            ParameterName_as8    := 'Output Cfg 29',
            ParameterType_u8     := 7,
            attr1_u              := 0,
            attr2_u              := 2,
            UnitCode_au8         := 0,
            AccesslevelCode_u8   := 129,
            attr4_u              := 0,
            EEPROMAddress_s      := (Page_u8 := 3, IntIndex_u8 := 92)
         ),

         (*********************************************)
         (* parameter 2.4.6 *)
         (*********************************************)
         (
            ParameterName_as8    := 'Output Cfg 30',
            ParameterType_u8     := 7,
            attr1_u              := 0,
            attr2_u              := 2,
            UnitCode_au8         := 0,
            AccesslevelCode_u8   := 129,
            attr4_u              := 0,
            EEPROMAddress_s      := (Page_u8 := 3, IntIndex_u8 := 93)
         ),

         (*********************************************)
         (* parameter 2.4.7 *)
         (*********************************************)
         (
            ParameterName_as8    := 'Output Cfg 31',
            ParameterType_u8     := 7,
            attr1_u              := 0,
            attr2_u              := 2,
            UnitCode_au8         := 0,
            AccesslevelCode_u8   := 129,
            attr4_u              := 0,
            EEPROMAddress_s      := (Page_u8 := 3, IntIndex_u8 := 94)
         ),

         (*********************************************)
         (* parameter 2.4.8 *)
         (*********************************************)
         (
            ParameterName_as8    := 'Output Cfg 32',
            ParameterType_u8     := 7,
            attr1_u              := 0,
            attr2_u              := 2,
            UnitCode_au8         := 0,
            AccesslevelCode_u8   := 129,
            attr4_u              := 0,
            EEPROMAddress_s      := (Page_u8 := 3, IntIndex_u8 := 95)
         )

      ),

      (*********************************************)
      (* parameter group 2.5 - up to 8 parameters can be defined here *)
      (*********************************************)
      (
         GroupName_as8   := 'Output Cfg 33-40',

         Param_as        := 

         (*********************************************)
         (* parameter 2.5.1 *)
         (*********************************************)
         (
            ParameterName_as8    := 'Output Cfg 33',
            ParameterType_u8     := 7,
            attr1_u              := 2,
            attr2_u              := 2,
            UnitCode_au8         := 0,
            AccesslevelCode_u8   := 129,
            attr4_u              := 0,
            EEPROMAddress_s      := (Page_u8 := 3, IntIndex_u8 := 96)
         ),

         (*********************************************)
         (* parameter 2.5.2 *)
         (*********************************************)
         (
            ParameterName_as8    := 'Output Cfg 34',
            ParameterType_u8     := 7,
            attr1_u              := 2,
            attr2_u              := 2,
            UnitCode_au8         := 0,
            AccesslevelCode_u8   := 129,
            attr4_u              := 0,
            EEPROMAddress_s      := (Page_u8 := 3, IntIndex_u8 := 97)
         ),

         (*********************************************)
         (* parameter 2.5.3 *)
         (*********************************************)
         (
            ParameterName_as8    := 'Output Cfg 35',
            ParameterType_u8     := 7,
            attr1_u              := 2,
            attr2_u              := 2,
            UnitCode_au8         := 0,
            AccesslevelCode_u8   := 129,
            attr4_u              := 0,
            EEPROMAddress_s      := (Page_u8 := 3, IntIndex_u8 := 98)
         ),

         (*********************************************)
         (* parameter 2.5.4 *)
         (*********************************************)
         (
            ParameterName_as8    := 'Output Cfg 36',
            ParameterType_u8     := 7,
            attr1_u              := 2,
            attr2_u              := 2,
            UnitCode_au8         := 0,
            AccesslevelCode_u8   := 129,
            attr4_u              := 0,
            EEPROMAddress_s      := (Page_u8 := 3, IntIndex_u8 := 99)
         ),

         (*********************************************)
         (* parameter 2.5.5 *)
         (*********************************************)
         (
            ParameterName_as8    := 'Output Cfg 37',
            ParameterType_u8     := 7,
            attr1_u              := 1,
            attr2_u              := 2,
            UnitCode_au8         := 0,
            AccesslevelCode_u8   := 129,
            attr4_u              := 0,
            EEPROMAddress_s      := (Page_u8 := 3, IntIndex_u8 := 100)
         ),

         (*********************************************)
         (* parameter 2.5.6 *)
         (*********************************************)
         (
            ParameterName_as8    := 'Output Cfg 38',
            ParameterType_u8     := 7,
            attr1_u              := 1,
            attr2_u              := 2,
            UnitCode_au8         := 0,
            AccesslevelCode_u8   := 129,
            attr4_u              := 0,
            EEPROMAddress_s      := (Page_u8 := 3, IntIndex_u8 := 101)
         ),

         (*********************************************)
         (* parameter 2.5.7 *)
         (*********************************************)
         (
            ParameterName_as8    := 'Output Cfg 39',
            ParameterType_u8     := 7,
            attr1_u              := 1,
            attr2_u              := 2,
            UnitCode_au8         := 0,
            AccesslevelCode_u8   := 129,
            attr4_u              := 0,
            EEPROMAddress_s      := (Page_u8 := 3, IntIndex_u8 := 102)
         ),

         (*********************************************)
         (* parameter 2.5.8 *)
         (*********************************************)
         (
            ParameterName_as8    := 'Output Cfg 40',
            ParameterType_u8     := 7,
            attr1_u              := 1,
            attr2_u              := 2,
            UnitCode_au8         := 0,
            AccesslevelCode_u8   := 129,
            attr4_u              := 0,
            EEPROMAddress_s      := (Page_u8 := 3, IntIndex_u8 := 103)
         )

      ),

      (*********************************************)
      (* parameter group 2.6 - up to 8 parameters can be defined here *)
      (*********************************************)
      (
         GroupName_as8   := 'Output Cfg 41-47',

         Param_as        := 

         (*********************************************)
         (* parameter 2.6.1 *)
         (*********************************************)
         (
            ParameterName_as8    := 'Output Cfg 41',
            ParameterType_u8     := 7,
            attr1_u              := 1,
            attr2_u              := 2,
            UnitCode_au8         := 0,
            AccesslevelCode_u8   := 129,
            attr4_u              := 0,
            EEPROMAddress_s      := (Page_u8 := 3, IntIndex_u8 := 104)
         ),

         (*********************************************)
         (* parameter 2.6.2 *)
         (*********************************************)
         (
            ParameterName_as8    := 'Output Cfg 42',
            ParameterType_u8     := 7,
            attr1_u              := 1,
            attr2_u              := 2,
            UnitCode_au8         := 0,
            AccesslevelCode_u8   := 129,
            attr4_u              := 0,
            EEPROMAddress_s      := (Page_u8 := 3, IntIndex_u8 := 105)
         ),

         (*********************************************)
         (* parameter 2.6.3 *)
         (*********************************************)
         (
            ParameterName_as8    := 'Output Cfg 43',
            ParameterType_u8     := 7,
            attr1_u              := 1,
            attr2_u              := 2,
            UnitCode_au8         := 0,
            AccesslevelCode_u8   := 129,
            attr4_u              := 0,
            EEPROMAddress_s      := (Page_u8 := 3, IntIndex_u8 := 106)
         ),

         (*********************************************)
         (* parameter 2.6.4 *)
         (*********************************************)
         (
            ParameterName_as8    := 'Output Cfg 44',
            ParameterType_u8     := 7,
            attr1_u              := 1,
            attr2_u              := 2,
            UnitCode_au8         := 0,
            AccesslevelCode_u8   := 129,
            attr4_u              := 0,
            EEPROMAddress_s      := (Page_u8 := 3, IntIndex_u8 := 107)
         ),

         (*********************************************)
         (* parameter 2.6.5 *)
         (*********************************************)
         (
            ParameterName_as8    := 'Output Cfg 45',
            ParameterType_u8     := 7,
            attr1_u              := 1,
            attr2_u              := 2,
            UnitCode_au8         := 0,
            AccesslevelCode_u8   := 129,
            attr4_u              := 0,
            EEPROMAddress_s      := (Page_u8 := 3, IntIndex_u8 := 108)
         ),

         (*********************************************)
         (* parameter 2.6.6 *)
         (*********************************************)
         (
            ParameterName_as8    := 'Output Cfg 46',
            ParameterType_u8     := 7,
            attr1_u              := 1,
            attr2_u              := 2,
            UnitCode_au8         := 0,
            AccesslevelCode_u8   := 129,
            attr4_u              := 0,
            EEPROMAddress_s      := (Page_u8 := 3, IntIndex_u8 := 109)
         ),

         (*********************************************)
         (* parameter 2.6.7 *)
         (*********************************************)
         (
            ParameterName_as8    := 'Output Cfg 47',
            ParameterType_u8     := 7,
            attr1_u              := 3,
            attr2_u              := 2,
            UnitCode_au8         := 0,
            AccesslevelCode_u8   := 129,
            attr4_u              := 1,
            EEPROMAddress_s      := (Page_u8 := 3, IntIndex_u8 := 110)
         ),

         (*********************************************)
         (* parameter 2.6.8 *)
         (*********************************************)
         (
         )

      ),

      (*********************************************)
      (* parameter group 2.7 - up to 8 parameters can be defined here *)
      (*********************************************)
      (
         GroupName_as8   := 'AOV Configuration',

         Param_as        := 

         (*********************************************)
         (* parameter 2.7.1 *)
         (*********************************************)
         (
            ParameterName_as8    := 'AOV Debounce',
            ParameterType_u8     := 0,
            attr1_u              := 50,
            attr2_u              := 250,
            attr3_u              := 10,
            UnitCode_au8         := 4,
            Multiplier_s16       := 1,
            Divisor_s16          := 1,
            NumberOfDigits_u16   := 0,
            AccesslevelCode_u8   := 179,
            attr4_u              := 200,
            EEPROMAddress_s      := (Page_u8 := 3, IntIndex_u8 := 112)
         ),

         (*********************************************)
         (* parameter 2.7.2 *)
         (*********************************************)
         (
            ParameterName_as8    := 'AOV Frequency',
            ParameterType_u8     := 0,
            attr1_u              := 0,
            attr2_u              := 5000,
            attr3_u              := 10,
            UnitCode_au8         := 0,
            Multiplier_s16       := 1,
            Divisor_s16          := 1,
            NumberOfDigits_u16   := 0,
            AccesslevelCode_u8   := 179,
            attr4_u              := 80,
            EEPROMAddress_s      := (Page_u8 := 3, IntIndex_u8 := 113)
         ),

         (*********************************************)
         (* parameter 2.7.3 *)
         (*********************************************)
         (
            ParameterName_as8    := 'AOV Resistance Min',
            ParameterType_u8     := 0,
            attr1_u              := 0,
            attr2_u              := 3000,
            attr3_u              := 10,
            UnitCode_au8         := 18,
            Multiplier_s16       := 1,
            Divisor_s16          := 1,
            NumberOfDigits_u16   := 0,
            AccesslevelCode_u8   := 179,
            attr4_u              := 0,
            EEPROMAddress_s      := (Page_u8 := 3, IntIndex_u8 := 114)
         ),

         (*********************************************)
         (* parameter 2.7.4 *)
         (*********************************************)
         (
            ParameterName_as8    := 'AOV Resistance Max',
            ParameterType_u8     := 0,
            attr1_u              := 0,
            attr2_u              := 3000,
            attr3_u              := 10,
            UnitCode_au8         := 18,
            Multiplier_s16       := 1,
            Divisor_s16          := 1,
            NumberOfDigits_u16   := 0,
            AccesslevelCode_u8   := 179,
            attr4_u              := 0,
            EEPROMAddress_s      := (Page_u8 := 3, IntIndex_u8 := 115)
         ),

         (*********************************************)
         (* parameter 2.7.5 *)
         (*********************************************)
         (
            ParameterName_as8    := 'AOV Kp',
            ParameterType_u8     := 0,
            attr1_u              := 0,
            attr2_u              := 2000,
            attr3_u              := 50,
            UnitCode_au8         := 0,
            Multiplier_s16       := 1,
            Divisor_s16          := 1,
            NumberOfDigits_u16   := 0,
            AccesslevelCode_u8   := 179,
            attr4_u              := 250,
            EEPROMAddress_s      := (Page_u8 := 3, IntIndex_u8 := 116)
         ),

         (*********************************************)
         (* parameter 2.7.6 *)
         (*********************************************)
         (
            ParameterName_as8    := 'AOV Ki',
            ParameterType_u8     := 0,
            attr1_u              := 0,
            attr2_u              := 500,
            attr3_u              := 50,
            UnitCode_au8         := 0,
            Multiplier_s16       := 1,
            Divisor_s16          := 1,
            NumberOfDigits_u16   := 0,
            AccesslevelCode_u8   := 179,
            attr4_u              := 250,
            EEPROMAddress_s      := (Page_u8 := 3, IntIndex_u8 := 117)
         ),

         (*********************************************)
         (* parameter 2.7.7 *)
         (*********************************************)
         (
         ),

         (*********************************************)
         (* parameter 2.7.8 *)
         (*********************************************)
         (
         )

      ),

      (*********************************************)
      (* parameter group 2.8 - up to 8 parameters can be defined here *)
      (*********************************************)
      (
         GroupName_as8   := 'AOC Configuration',

         Param_as        := 

         (*********************************************)
         (* parameter 2.8.1 *)
         (*********************************************)
         (
            ParameterName_as8    := 'AOC Debounce',
            ParameterType_u8     := 0,
            attr1_u              := 50,
            attr2_u              := 250,
            attr3_u              := 10,
            UnitCode_au8         := 4,
            Multiplier_s16       := 1,
            Divisor_s16          := 1,
            NumberOfDigits_u16   := 0,
            AccesslevelCode_u8   := 179,
            attr4_u              := 200,
            EEPROMAddress_s      := (Page_u8 := 3, IntIndex_u8 := 120)
         ),

         (*********************************************)
         (* parameter 2.8.2 *)
         (*********************************************)
         (
            ParameterName_as8    := 'AOC Frequency',
            ParameterType_u8     := 0,
            attr1_u              := 0,
            attr2_u              := 5000,
            attr3_u              := 10,
            UnitCode_au8         := 0,
            AccesslevelCode_u8   := 179,
            attr4_u              := 5000,
            EEPROMAddress_s      := (Page_u8 := 3, IntIndex_u8 := 121)
         ),

         (*********************************************)
         (* parameter 2.8.3 *)
         (*********************************************)
         (
            ParameterName_as8    := 'AOC Resistance Min',
            ParameterType_u8     := 0,
            attr1_u              := 0,
            attr2_u              := 3000,
            attr3_u              := 10,
            UnitCode_au8         := 18,
            Multiplier_s16       := 1,
            Divisor_s16          := 1,
            NumberOfDigits_u16   := 0,
            AccesslevelCode_u8   := 179,
            attr4_u              := 0,
            EEPROMAddress_s      := (Page_u8 := 3, IntIndex_u8 := 122)
         ),

         (*********************************************)
         (* parameter 2.8.4 *)
         (*********************************************)
         (
            ParameterName_as8    := 'AOC Resistance Max',
            ParameterType_u8     := 0,
            attr1_u              := 0,
            attr2_u              := 3000,
            attr3_u              := 10,
            UnitCode_au8         := 18,
            Multiplier_s16       := 1,
            Divisor_s16          := 1,
            NumberOfDigits_u16   := 0,
            AccesslevelCode_u8   := 179,
            attr4_u              := 0,
            EEPROMAddress_s      := (Page_u8 := 3, IntIndex_u8 := 123)
         ),

         (*********************************************)
         (* parameter 2.8.5 *)
         (*********************************************)
         (
            ParameterName_as8    := 'AOC Kp',
            ParameterType_u8     := 0,
            attr1_u              := 0,
            attr2_u              := 2000,
            attr3_u              := 50,
            UnitCode_au8         := 0,
            Multiplier_s16       := 1,
            Divisor_s16          := 1,
            NumberOfDigits_u16   := 0,
            AccesslevelCode_u8   := 179,
            attr4_u              := 250,
            EEPROMAddress_s      := (Page_u8 := 3, IntIndex_u8 := 124)
         ),

         (*********************************************)
         (* parameter 2.8.6 *)
         (*********************************************)
         (
            ParameterName_as8    := 'AOC Ki',
            ParameterType_u8     := 0,
            attr1_u              := 0,
            attr2_u              := 500,
            attr3_u              := 50,
            UnitCode_au8         := 0,
            Multiplier_s16       := 1,
            Divisor_s16          := 1,
            NumberOfDigits_u16   := 0,
            AccesslevelCode_u8   := 179,
            attr4_u              := 250,
            EEPROMAddress_s      := (Page_u8 := 3, IntIndex_u8 := 125)
         ),

         (*********************************************)
         (* parameter 2.8.7 *)
         (*********************************************)
         (
         ),

         (*********************************************)
         (* parameter 2.8.8 *)
         (*********************************************)
         (
         )

      )

   ),

   (*********************************************)
   (* parameter menu 3 - up to 8 groups can be defined here *)
   (*********************************************)
   (
      MenuName_as8        := 'Menu 3',

      ParameterGroup_as   := 

      (*********************************************)
      (* parameter group 3.1 - up to 8 parameters can be defined here *)
      (*********************************************)
      (
         GroupName_as8   := 'Output Value 1-8',

         Param_as        := 

         (*********************************************)
         (* parameter 3.1.1 *)
         (*********************************************)
         (
            ParameterName_as8    := 'Output Value 1',
            ParameterType_u8     := 0,
            attr1_u              := 0,
            attr2_u              := 10000,
            attr3_u              := 50,
            UnitCode_au8         := 15,
            Multiplier_s16       := 1,
            Divisor_s16          := 1,
            NumberOfDigits_u16   := 0,
            AccesslevelCode_u8   := 129,
            attr4_u              := 0,
            EEPROMAddress_s      := (Page_u8 := 3, IntIndex_u8 := 128)
         ),

         (*********************************************)
         (* parameter 3.1.2 *)
         (*********************************************)
         (
            ParameterName_as8    := 'Output Value 2',
            ParameterType_u8     := 0,
            attr1_u              := 0,
            attr2_u              := 10000,
            attr3_u              := 50,
            UnitCode_au8         := 15,
            Multiplier_s16       := 1,
            Divisor_s16          := 1,
            NumberOfDigits_u16   := 0,
            AccesslevelCode_u8   := 129,
            attr4_u              := 0,
            EEPROMAddress_s      := (Page_u8 := 3, IntIndex_u8 := 129)
         ),

         (*********************************************)
         (* parameter 3.1.3 *)
         (*********************************************)
         (
            ParameterName_as8    := 'Output Value 3',
            ParameterType_u8     := 0,
            attr1_u              := 0,
            attr2_u              := 10000,
            attr3_u              := 50,
            UnitCode_au8         := 15,
            Multiplier_s16       := 1,
            Divisor_s16          := 1,
            NumberOfDigits_u16   := 0,
            AccesslevelCode_u8   := 129,
            attr4_u              := 0,
            EEPROMAddress_s      := (Page_u8 := 3, IntIndex_u8 := 130)
         ),

         (*********************************************)
         (* parameter 3.1.4 *)
         (*********************************************)
         (
            ParameterName_as8    := 'Output Value 4',
            ParameterType_u8     := 0,
            attr1_u              := 0,
            attr2_u              := 10000,
            attr3_u              := 50,
            UnitCode_au8         := 15,
            Multiplier_s16       := 1,
            Divisor_s16          := 1,
            NumberOfDigits_u16   := 0,
            AccesslevelCode_u8   := 129,
            attr4_u              := 0,
            EEPROMAddress_s      := (Page_u8 := 3, IntIndex_u8 := 131)
         ),

         (*********************************************)
         (* parameter 3.1.5 *)
         (*********************************************)
         (
            ParameterName_as8    := 'Output Value 5',
            ParameterType_u8     := 0,
            attr1_u              := 0,
            attr2_u              := 10000,
            attr3_u              := 50,
            UnitCode_au8         := 15,
            Multiplier_s16       := 1,
            Divisor_s16          := 1,
            NumberOfDigits_u16   := 0,
            AccesslevelCode_u8   := 129,
            attr4_u              := 0,
            EEPROMAddress_s      := (Page_u8 := 3, IntIndex_u8 := 132)
         ),

         (*********************************************)
         (* parameter 3.1.6 *)
         (*********************************************)
         (
            ParameterName_as8    := 'Output Value 6',
            ParameterType_u8     := 0,
            attr1_u              := 0,
            attr2_u              := 10000,
            attr3_u              := 50,
            UnitCode_au8         := 15,
            Multiplier_s16       := 1,
            Divisor_s16          := 1,
            NumberOfDigits_u16   := 0,
            AccesslevelCode_u8   := 129,
            attr4_u              := 0,
            EEPROMAddress_s      := (Page_u8 := 3, IntIndex_u8 := 133)
         ),

         (*********************************************)
         (* parameter 3.1.7 *)
         (*********************************************)
         (
            ParameterName_as8    := 'Output Value 7',
            ParameterType_u8     := 0,
            attr1_u              := 0,
            attr2_u              := 10000,
            attr3_u              := 50,
            UnitCode_au8         := 15,
            Multiplier_s16       := 1,
            Divisor_s16          := 1,
            NumberOfDigits_u16   := 0,
            AccesslevelCode_u8   := 129,
            attr4_u              := 0,
            EEPROMAddress_s      := (Page_u8 := 3, IntIndex_u8 := 134)
         ),

         (*********************************************)
         (* parameter 3.1.8 *)
         (*********************************************)
         (
            ParameterName_as8    := 'Output Value 8',
            ParameterType_u8     := 0,
            attr1_u              := 0,
            attr2_u              := 10000,
            attr3_u              := 50,
            UnitCode_au8         := 15,
            Multiplier_s16       := 1,
            Divisor_s16          := 1,
            NumberOfDigits_u16   := 0,
            AccesslevelCode_u8   := 129,
            attr4_u              := 0,
            EEPROMAddress_s      := (Page_u8 := 3, IntIndex_u8 := 135)
         )

      ),

      (*********************************************)
      (* parameter group 3.2 - up to 8 parameters can be defined here *)
      (*********************************************)
      (
         GroupName_as8   := 'Output Value 9-16',

         Param_as        := 

         (*********************************************)
         (* parameter 3.2.1 *)
         (*********************************************)
         (
            ParameterName_as8    := 'Output Value 9',
            ParameterType_u8     := 0,
            attr1_u              := 0,
            attr2_u              := 10000,
            attr3_u              := 50,
            UnitCode_au8         := 15,
            Multiplier_s16       := 1,
            Divisor_s16          := 1,
            NumberOfDigits_u16   := 0,
            AccesslevelCode_u8   := 129,
            attr4_u              := 0,
            EEPROMAddress_s      := (Page_u8 := 3, IntIndex_u8 := 136)
         ),

         (*********************************************)
         (* parameter 3.2.2 *)
         (*********************************************)
         (
            ParameterName_as8    := 'Output Value 10',
            ParameterType_u8     := 0,
            attr1_u              := 0,
            attr2_u              := 10000,
            attr3_u              := 50,
            UnitCode_au8         := 15,
            Multiplier_s16       := 1,
            Divisor_s16          := 1,
            NumberOfDigits_u16   := 0,
            AccesslevelCode_u8   := 129,
            attr4_u              := 0,
            EEPROMAddress_s      := (Page_u8 := 3, IntIndex_u8 := 137)
         ),

         (*********************************************)
         (* parameter 3.2.3 *)
         (*********************************************)
         (
            ParameterName_as8    := 'Output Value 11',
            ParameterType_u8     := 0,
            attr1_u              := 0,
            attr2_u              := 10000,
            attr3_u              := 50,
            UnitCode_au8         := 15,
            Multiplier_s16       := 1,
            Divisor_s16          := 1,
            NumberOfDigits_u16   := 0,
            AccesslevelCode_u8   := 129,
            attr4_u              := 0,
            EEPROMAddress_s      := (Page_u8 := 3, IntIndex_u8 := 138)
         ),

         (*********************************************)
         (* parameter 3.2.4 *)
         (*********************************************)
         (
            ParameterName_as8    := 'Output Value 12',
            ParameterType_u8     := 0,
            attr1_u              := 0,
            attr2_u              := 10000,
            attr3_u              := 50,
            UnitCode_au8         := 15,
            Multiplier_s16       := 1,
            Divisor_s16          := 1,
            NumberOfDigits_u16   := 0,
            AccesslevelCode_u8   := 129,
            attr4_u              := 0,
            EEPROMAddress_s      := (Page_u8 := 3, IntIndex_u8 := 139)
         ),

         (*********************************************)
         (* parameter 3.2.5 *)
         (*********************************************)
         (
            ParameterName_as8    := 'Output Value 13',
            ParameterType_u8     := 0,
            attr1_u              := 0,
            attr2_u              := 10000,
            attr3_u              := 50,
            UnitCode_au8         := 15,
            Multiplier_s16       := 1,
            Divisor_s16          := 1,
            NumberOfDigits_u16   := 0,
            AccesslevelCode_u8   := 129,
            attr4_u              := 0,
            EEPROMAddress_s      := (Page_u8 := 3, IntIndex_u8 := 140)
         ),

         (*********************************************)
         (* parameter 3.2.6 *)
         (*********************************************)
         (
            ParameterName_as8    := 'Output Value 14',
            ParameterType_u8     := 0,
            attr1_u              := 0,
            attr2_u              := 10000,
            attr3_u              := 50,
            UnitCode_au8         := 15,
            Multiplier_s16       := 1,
            Divisor_s16          := 1,
            NumberOfDigits_u16   := 0,
            AccesslevelCode_u8   := 129,
            attr4_u              := 0,
            EEPROMAddress_s      := (Page_u8 := 3, IntIndex_u8 := 141)
         ),

         (*********************************************)
         (* parameter 3.2.7 *)
         (*********************************************)
         (
            ParameterName_as8    := 'Output Value 15',
            ParameterType_u8     := 0,
            attr1_u              := 0,
            attr2_u              := 10000,
            attr3_u              := 50,
            UnitCode_au8         := 15,
            Multiplier_s16       := 1,
            Divisor_s16          := 1,
            NumberOfDigits_u16   := 0,
            AccesslevelCode_u8   := 129,
            attr4_u              := 0,
            EEPROMAddress_s      := (Page_u8 := 3, IntIndex_u8 := 142)
         ),

         (*********************************************)
         (* parameter 3.2.8 *)
         (*********************************************)
         (
            ParameterName_as8    := 'Output Value 16',
            ParameterType_u8     := 0,
            attr1_u              := 0,
            attr2_u              := 10000,
            attr3_u              := 50,
            UnitCode_au8         := 15,
            Multiplier_s16       := 1,
            Divisor_s16          := 1,
            NumberOfDigits_u16   := 0,
            AccesslevelCode_u8   := 129,
            attr4_u              := 0,
            EEPROMAddress_s      := (Page_u8 := 3, IntIndex_u8 := 143)
         )

      ),

      (*********************************************)
      (* parameter group 3.3 - up to 8 parameters can be defined here *)
      (*********************************************)
      (
         GroupName_as8   := 'Output Value 17-36',

         Param_as        := 

         (*********************************************)
         (* parameter 3.3.1 *)
         (*********************************************)
         (
            ParameterName_as8    := 'Output Value 17',
            ParameterType_u8     := 0,
            attr1_u              := 0,
            attr2_u              := 10000,
            attr3_u              := 50,
            UnitCode_au8         := 15,
            Multiplier_s16       := 1,
            Divisor_s16          := 1,
            NumberOfDigits_u16   := 0,
            AccesslevelCode_u8   := 129,
            attr4_u              := 0,
            EEPROMAddress_s      := (Page_u8 := 3, IntIndex_u8 := 144)
         ),

         (*********************************************)
         (* parameter 3.3.2 *)
         (*********************************************)
         (
            ParameterName_as8    := 'Output Value 18',
            ParameterType_u8     := 0,
            attr1_u              := 0,
            attr2_u              := 10000,
            attr3_u              := 50,
            UnitCode_au8         := 15,
            Multiplier_s16       := 1,
            Divisor_s16          := 1,
            NumberOfDigits_u16   := 0,
            AccesslevelCode_u8   := 129,
            attr4_u              := 0,
            EEPROMAddress_s      := (Page_u8 := 3, IntIndex_u8 := 145)
         ),

         (*********************************************)
         (* parameter 3.3.3 *)
         (*********************************************)
         (
         ),

         (*********************************************)
         (* parameter 3.3.4 *)
         (*********************************************)
         (
         ),

         (*********************************************)
         (* parameter 3.3.5 *)
         (*********************************************)
         (
            ParameterName_as8    := 'Output Value 33',
            ParameterType_u8     := 0,
            attr1_u              := 0,
            attr2_u              := 10000,
            attr3_u              := 50,
            UnitCode_au8         := 15,
            Multiplier_s16       := 1,
            Divisor_s16          := 1,
            NumberOfDigits_u16   := 0,
            AccesslevelCode_u8   := 129,
            attr4_u              := 0,
            EEPROMAddress_s      := (Page_u8 := 3, IntIndex_u8 := 148)
         ),

         (*********************************************)
         (* parameter 3.3.6 *)
         (*********************************************)
         (
            ParameterName_as8    := 'Output Value 34',
            ParameterType_u8     := 0,
            attr1_u              := 0,
            attr2_u              := 10000,
            attr3_u              := 50,
            UnitCode_au8         := 15,
            Multiplier_s16       := 1,
            Divisor_s16          := 1,
            NumberOfDigits_u16   := 0,
            AccesslevelCode_u8   := 129,
            attr4_u              := 0,
            EEPROMAddress_s      := (Page_u8 := 3, IntIndex_u8 := 149)
         ),

         (*********************************************)
         (* parameter 3.3.7 *)
         (*********************************************)
         (
            ParameterName_as8    := 'Output Value 35',
            ParameterType_u8     := 0,
            attr1_u              := 0,
            attr2_u              := 10000,
            attr3_u              := 50,
            UnitCode_au8         := 15,
            Multiplier_s16       := 1,
            Divisor_s16          := 1,
            NumberOfDigits_u16   := 0,
            AccesslevelCode_u8   := 129,
            attr4_u              := 0,
            EEPROMAddress_s      := (Page_u8 := 3, IntIndex_u8 := 150)
         ),

         (*********************************************)
         (* parameter 3.3.8 *)
         (*********************************************)
         (
            ParameterName_as8    := 'Output Value 36',
            ParameterType_u8     := 0,
            attr1_u              := 0,
            attr2_u              := 10000,
            attr3_u              := 50,
            UnitCode_au8         := 15,
            Multiplier_s16       := 1,
            Divisor_s16          := 1,
            NumberOfDigits_u16   := 0,
            AccesslevelCode_u8   := 129,
            attr4_u              := 0,
            EEPROMAddress_s      := (Page_u8 := 3, IntIndex_u8 := 151)
         )

      ),

      (*********************************************)
      (* parameter group 3.4 - up to 8 parameters can be defined here *)
      (*********************************************)
      (
         GroupName_as8   := 'Output Value 37-44',

         Param_as        := 

         (*********************************************)
         (* parameter 3.4.1 *)
         (*********************************************)
         (
            ParameterName_as8    := 'Output Value 37',
            ParameterType_u8     := 0,
            attr1_u              := 0,
            attr2_u              := 10000,
            attr3_u              := 50,
            UnitCode_au8         := 15,
            Multiplier_s16       := 1,
            Divisor_s16          := 1,
            NumberOfDigits_u16   := 0,
            AccesslevelCode_u8   := 129,
            attr4_u              := 0,
            EEPROMAddress_s      := (Page_u8 := 3, IntIndex_u8 := 152)
         ),

         (*********************************************)
         (* parameter 3.4.2 *)
         (*********************************************)
         (
            ParameterName_as8    := 'Output Value 38',
            ParameterType_u8     := 0,
            attr1_u              := 0,
            attr2_u              := 10000,
            attr3_u              := 50,
            UnitCode_au8         := 15,
            Multiplier_s16       := 1,
            Divisor_s16          := 1,
            NumberOfDigits_u16   := 0,
            AccesslevelCode_u8   := 129,
            attr4_u              := 0,
            EEPROMAddress_s      := (Page_u8 := 3, IntIndex_u8 := 153)
         ),

         (*********************************************)
         (* parameter 3.4.3 *)
         (*********************************************)
         (
            ParameterName_as8    := 'Output Value 39',
            ParameterType_u8     := 0,
            attr1_u              := 0,
            attr2_u              := 10000,
            attr3_u              := 50,
            UnitCode_au8         := 15,
            Multiplier_s16       := 1,
            Divisor_s16          := 1,
            NumberOfDigits_u16   := 0,
            AccesslevelCode_u8   := 129,
            attr4_u              := 0,
            EEPROMAddress_s      := (Page_u8 := 3, IntIndex_u8 := 154)
         ),

         (*********************************************)
         (* parameter 3.4.4 *)
         (*********************************************)
         (
            ParameterName_as8    := 'Output Value 40',
            ParameterType_u8     := 0,
            attr1_u              := 0,
            attr2_u              := 10000,
            attr3_u              := 50,
            UnitCode_au8         := 15,
            Multiplier_s16       := 1,
            Divisor_s16          := 1,
            NumberOfDigits_u16   := 0,
            AccesslevelCode_u8   := 129,
            attr4_u              := 0,
            EEPROMAddress_s      := (Page_u8 := 3, IntIndex_u8 := 155)
         ),

         (*********************************************)
         (* parameter 3.4.5 *)
         (*********************************************)
         (
            ParameterName_as8    := 'Output Value 41',
            ParameterType_u8     := 0,
            attr1_u              := 0,
            attr2_u              := 10000,
            attr3_u              := 50,
            UnitCode_au8         := 15,
            Multiplier_s16       := 1,
            Divisor_s16          := 1,
            NumberOfDigits_u16   := 0,
            AccesslevelCode_u8   := 129,
            attr4_u              := 0,
            EEPROMAddress_s      := (Page_u8 := 3, IntIndex_u8 := 156)
         ),

         (*********************************************)
         (* parameter 3.4.6 *)
         (*********************************************)
         (
            ParameterName_as8    := 'Output Value 42',
            ParameterType_u8     := 0,
            attr1_u              := 0,
            attr2_u              := 10000,
            attr3_u              := 50,
            UnitCode_au8         := 15,
            Multiplier_s16       := 1,
            Divisor_s16          := 1,
            NumberOfDigits_u16   := 0,
            AccesslevelCode_u8   := 129,
            attr4_u              := 0,
            EEPROMAddress_s      := (Page_u8 := 3, IntIndex_u8 := 157)
         ),

         (*********************************************)
         (* parameter 3.4.7 *)
         (*********************************************)
         (
            ParameterName_as8    := 'Output Value 43',
            ParameterType_u8     := 0,
            attr1_u              := 0,
            attr2_u              := 10000,
            attr3_u              := 50,
            UnitCode_au8         := 15,
            Multiplier_s16       := 1,
            Divisor_s16          := 1,
            NumberOfDigits_u16   := 0,
            AccesslevelCode_u8   := 129,
            attr4_u              := 0,
            EEPROMAddress_s      := (Page_u8 := 3, IntIndex_u8 := 158)
         ),

         (*********************************************)
         (* parameter 3.4.8 *)
         (*********************************************)
         (
            ParameterName_as8    := 'Output Value 44',
            ParameterType_u8     := 0,
            attr1_u              := 0,
            attr2_u              := 10000,
            attr3_u              := 50,
            UnitCode_au8         := 15,
            Multiplier_s16       := 1,
            Divisor_s16          := 1,
            NumberOfDigits_u16   := 0,
            AccesslevelCode_u8   := 129,
            attr4_u              := 0,
            EEPROMAddress_s      := (Page_u8 := 3, IntIndex_u8 := 159)
         )

      ),

      (*********************************************)
      (* parameter group 3.5 - up to 8 parameters can be defined here *)
      (*********************************************)
      (
         GroupName_as8   := 'Output Value 45-47',

         Param_as        := 

         (*********************************************)
         (* parameter 3.5.1 *)
         (*********************************************)
         (
            ParameterName_as8    := 'Output Value 45',
            ParameterType_u8     := 0,
            attr1_u              := 0,
            attr2_u              := 10000,
            attr3_u              := 50,
            UnitCode_au8         := 15,
            Multiplier_s16       := 1,
            Divisor_s16          := 1,
            NumberOfDigits_u16   := 0,
            AccesslevelCode_u8   := 129,
            attr4_u              := 0,
            EEPROMAddress_s      := (Page_u8 := 3, IntIndex_u8 := 160)
         ),

         (*********************************************)
         (* parameter 3.5.2 *)
         (*********************************************)
         (
            ParameterName_as8    := 'Output Value 46',
            ParameterType_u8     := 0,
            attr1_u              := 0,
            attr2_u              := 10000,
            attr3_u              := 50,
            UnitCode_au8         := 15,
            Multiplier_s16       := 1,
            Divisor_s16          := 1,
            NumberOfDigits_u16   := 0,
            AccesslevelCode_u8   := 129,
            attr4_u              := 0,
            EEPROMAddress_s      := (Page_u8 := 3, IntIndex_u8 := 161)
         ),

         (*********************************************)
         (* parameter 3.5.3 *)
         (*********************************************)
         (
            ParameterName_as8    := 'Output Value 47',
            ParameterType_u8     := 0,
            attr1_u              := 0,
            attr2_u              := 20000,
            attr3_u              := 50,
            UnitCode_au8         := 15,
            Multiplier_s16       := 1,
            Divisor_s16          := 1,
            NumberOfDigits_u16   := 0,
            AccesslevelCode_u8   := 129,
            attr4_u              := 0,
            EEPROMAddress_s      := (Page_u8 := 3, IntIndex_u8 := 162)
         ),

         (*********************************************)
         (* parameter 3.5.4 *)
         (*********************************************)
         (
         ),

         (*********************************************)
         (* parameter 3.5.5 *)
         (*********************************************)
         (
         ),

         (*********************************************)
         (* parameter 3.5.6 *)
         (*********************************************)
         (
         ),

         (*********************************************)
         (* parameter 3.5.7 *)
         (*********************************************)
         (
         ),

         (*********************************************)
         (* parameter 3.5.8 *)
         (*********************************************)
         (
         )

      ),

      (*********************************************)
      (* parameter group 3.6 - up to 8 parameters can be defined here *)
      (*********************************************)
      (
         GroupName_as8   := 'POH Configuration',

         Param_as        := 

         (*********************************************)
         (* parameter 3.6.1 *)
         (*********************************************)
         (
            ParameterName_as8    := 'POH Debounce',
            ParameterType_u8     := 0,
            attr1_u              := 50,
            attr2_u              := 250,
            attr3_u              := 10,
            UnitCode_au8         := 4,
            Multiplier_s16       := 1,
            Divisor_s16          := 1,
            NumberOfDigits_u16   := 0,
            AccesslevelCode_u8   := 179,
            attr4_u              := 100,
            EEPROMAddress_s      := (Page_u8 := 3, IntIndex_u8 := 168)
         ),

         (*********************************************)
         (* parameter 3.6.2 *)
         (*********************************************)
         (
         ),

         (*********************************************)
         (* parameter 3.6.3 *)
         (*********************************************)
         (
            ParameterName_as8    := 'POH Resistance Min',
            ParameterType_u8     := 0,
            attr1_u              := 0,
            attr2_u              := 3000,
            attr3_u              := 10,
            UnitCode_au8         := 18,
            Multiplier_s16       := 1,
            Divisor_s16          := 1,
            NumberOfDigits_u16   := 0,
            AccesslevelCode_u8   := 179,
            attr4_u              := 2,
            EEPROMAddress_s      := (Page_u8 := 3, IntIndex_u8 := 170)
         ),

         (*********************************************)
         (* parameter 3.6.4 *)
         (*********************************************)
         (
            ParameterName_as8    := 'POH Resistance Max',
            ParameterType_u8     := 0,
            attr1_u              := 0,
            attr2_u              := 3000,
            attr3_u              := 10,
            UnitCode_au8         := 18,
            Multiplier_s16       := 1,
            Divisor_s16          := 1,
            NumberOfDigits_u16   := 0,
            AccesslevelCode_u8   := 179,
            attr4_u              := 52,
            EEPROMAddress_s      := (Page_u8 := 3, IntIndex_u8 := 171)
         ),

         (*********************************************)
         (* parameter 3.6.5 *)
         (*********************************************)
         (
            ParameterName_as8    := 'POH Kp',
            ParameterType_u8     := 0,
            attr1_u              := 0,
            attr2_u              := 2000,
            attr3_u              := 50,
            UnitCode_au8         := 0,
            Multiplier_s16       := 1,
            Divisor_s16          := 1,
            NumberOfDigits_u16   := 0,
            AccesslevelCode_u8   := 179,
            attr4_u              := 250,
            EEPROMAddress_s      := (Page_u8 := 3, IntIndex_u8 := 172)
         ),

         (*********************************************)
         (* parameter 3.6.6 *)
         (*********************************************)
         (
            ParameterName_as8    := 'POH Ki',
            ParameterType_u8     := 0,
            attr1_u              := 0,
            attr2_u              := 500,
            attr3_u              := 50,
            UnitCode_au8         := 0,
            Multiplier_s16       := 1,
            Divisor_s16          := 1,
            NumberOfDigits_u16   := 0,
            AccesslevelCode_u8   := 179,
            attr4_u              := 250,
            EEPROMAddress_s      := (Page_u8 := 3, IntIndex_u8 := 173)
         ),

         (*********************************************)
         (* parameter 3.6.7 *)
         (*********************************************)
         (
         ),

         (*********************************************)
         (* parameter 3.6.8 *)
         (*********************************************)
         (
         )

      ),

      (*********************************************)
      (* parameter group 3.7 - up to 8 parameters can be defined here *)
      (*********************************************)
      (
         GroupName_as8   := 'POL Configuration',

         Param_as        := 

         (*********************************************)
         (* parameter 3.7.1 *)
         (*********************************************)
         (
            ParameterName_as8    := 'POL Debounce',
            ParameterType_u8     := 0,
            attr1_u              := 50,
            attr2_u              := 250,
            attr3_u              := 10,
            UnitCode_au8         := 4,
            Multiplier_s16       := 1,
            Divisor_s16          := 1,
            NumberOfDigits_u16   := 0,
            AccesslevelCode_u8   := 179,
            attr4_u              := 100,
            EEPROMAddress_s      := (Page_u8 := 3, IntIndex_u8 := 176)
         ),

         (*********************************************)
         (* parameter 3.7.2 *)
         (*********************************************)
         (
         ),

